(* CoDeSys 2.3 export: PLC_PRG.EXP *)

(* POU PLC_PRG, FBD *)
PROGRAM PLC_PRG
VAR
	ied1_modbus: IED_BLOCK;
	ied2_modbus: IED_BLOCK;
END_VAR
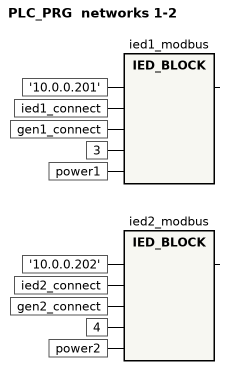
_FBD_ (* Function Block Diagram *)
NETWORK 1
	ied1_modbus:IED_BLOCK('10.0.0.201', ied1_connect, gen1_connect, 3, power1)
NETWORK 2
	ied2_modbus:IED_BLOCK('10.0.0.202', ied2_connect, gen2_connect, 4, power2)
_END_FBD_
(* the same logic as Structured Text *)
(* Network 1 *)
ied1_modbus('10.0.0.201', ied1_connect, gen1_connect, 3, power1);
(* Network 2 *)
ied2_modbus('10.0.0.202', ied2_connect, gen2_connect, 4, power2);
END_PROGRAM
